(* CODESYS project Test_Modbus_HMI.project
   Title: Test_Modbus_TCP_IP
   Version: 0.0.0.0
   Author: serbogr1

Project tree, tasks and I/O mapping:
  MyController : TM241CE40R, Schneider Electric, order no. TM241CE40R, version 4.0.6.18
    application Application
      task MAST (cyclic, interval 20 ms, priority 15, watchdog 100 ms x 1) calls MyPOU
      global variables GVL
      program MyPOU [ST]
      visualisation ModbusTCP
    DI : Digital Inputs, Schneider Electric, version 4.0.6.18
        input  idwDI_IDW0 : DWORD  // IDW0
        input  ibDI_IB1 : BYTE  // IB1
    DQ : Digital Outputs, Schneider Electric, version 4.0.6.18
        output qwDQ_QW0 : WORD  // QW0
        output qbDQ_QB1 : BYTE  // QB1
    Counters : Counters, Schneider Electric, version 4.0.6.18
    Pulse_Generators : Pulse Generators, Schneider Electric, version 4.0.6.18
    Cartridge_1 : Cartridge, Schneider Electric, version 4.0.6.18
    Cartridge_2 : Cartridge, Schneider Electric, version 4.0.6.18
    IO_Bus : IO bus - TM3, Schneider Electric, version 4.0.6.18
    COM_Bus : COM bus, Schneider Electric, version 4.0.6.18
    Ethernet_1 : Ethernet Network, Schneider Electric, version 4.0.6.18
        settings: IPAddress = [172, 16, 191, 108]; SubnetMask = [255, 255, 255, 0]; GatewayAddress = [172, 16, 191, 1]; WebServer = TRUE; FTP Server = TRUE; SoMachine Protocol = TRUE; Modbus Server = TRUE; NetManage Protocol = TRUE; SNMP protocol = TRUE; Enable Routing = FALSE; WebVisu protocol = TRUE; DHCP Server Active = FALSE
    Serial_Line_1 : Serial line, Schneider Electric, version 4.0.6.18
    Serial_Line_2 : Serial line, Schneider Electric, version 4.0.6.18
  text list GlobalTextList
*)

// MyController/Application/GVL
VAR_GLOBAL
END_VAR

// MyController/Application/MyPOU
PROGRAM MyPOU
VAR
	HMI_INPUT AT %MW100: WORD;
	HIMI_OUTPUT AT %MW110: WORD;
END_VAR

END_PROGRAM

// MyController/Application/ModbusTCP
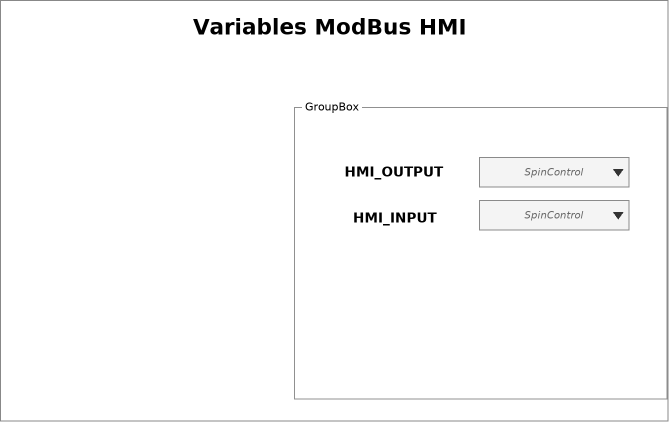
VISUALIZATION ModbusTCP  // 669x422
    Label (150,12 360x30), "Variables ModBus HMI"
    Label (57,115 150x30)
    GroupBox (294,99 373x300), "GroupBox"
        Label (25,58 150x30), "HMI_OUTPUT"
        Label (26,104 150x30), "HMI_INPUT"
        SpinControl (185,58 150x30), variable: MyPOU.HIMI_OUTPUT
        SpinControl (185,101 150x30), variable: MyPOU.HMI_INPUT
        Label (30,197 150x30)
        Label (31,245 150x30)
        Label (32,291 150x30)
END_VISUALIZATION
